// LS Electric XG5000 project: Villa 4 - ALS
// PLC NewPLC
// module base 0 slot 0: Input/Output Module:XBC-DR40S (DC 24V INPUT 24points/RELAY OUTPUT 16points)
// module base 0 slot 1: FEnet:XBL-EMTA

PROGRAM Main (task: Scan Program)

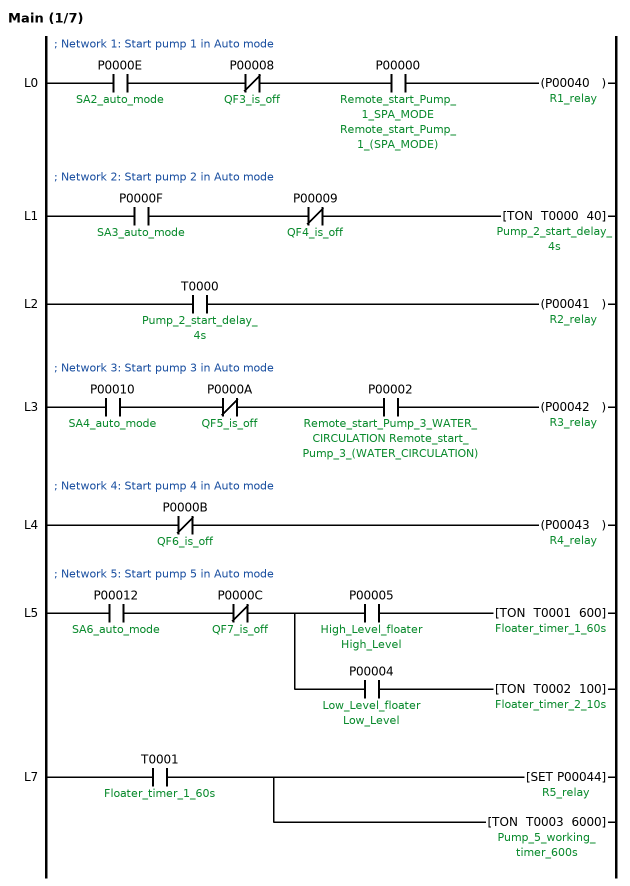
; L0
LOAD      P0000E	// SA2_auto_mode
AND NOT   P00008	// QF3_is_off
AND       P00000	// Remote_start_Pump_1_SPA_MODE Remote_start_Pump_1_(SPA_MODE)
OUT       P00040	// R1_relay
// output comment: Network 1: Start pump 1 in Auto mode
; L1
LOAD      P0000F	// SA3_auto_mode
AND NOT   P00009	// QF4_is_off
TON       T0000 40	// Pump_2_start_delay_4s
// output comment: Network 2: Start pump 2 in Auto mode
; L2
LOAD      T0000	// Pump_2_start_delay_4s
OUT       P00041	// R2_relay
; L3
LOAD      P00010	// SA4_auto_mode
AND NOT   P0000A	// QF5_is_off
AND       P00002	// Remote_start_Pump_3_WATER_CIRCULATION Remote_start_Pump_3_(WATER_CIRCULATION)
OUT       P00042	// R3_relay
// output comment: Network 3: Start pump 3 in Auto mode
; L4
LOAD NOT  P0000B	// QF6_is_off
OUT       P00043	// R4_relay
// output comment: Network 4: Start pump 4 in Auto mode
; L5
LOAD      P00012	// SA6_auto_mode
AND NOT   P0000C	// QF7_is_off
MPUSH
AND       P00005	// High_Level_floater High_Level
TON       T0001 600	// Floater_timer_1_60s
MPOP
AND       P00004	// Low_Level_floater Low_Level
TON       T0002 100	// Floater_timer_2_10s
// output comment: Network 5: Start pump 5 in Auto mode
; L7
LOAD      T0001	// Floater_timer_1_60s
SET       P00044	// R5_relay
TON       T0003 6000	// Pump_5_working_timer_600s

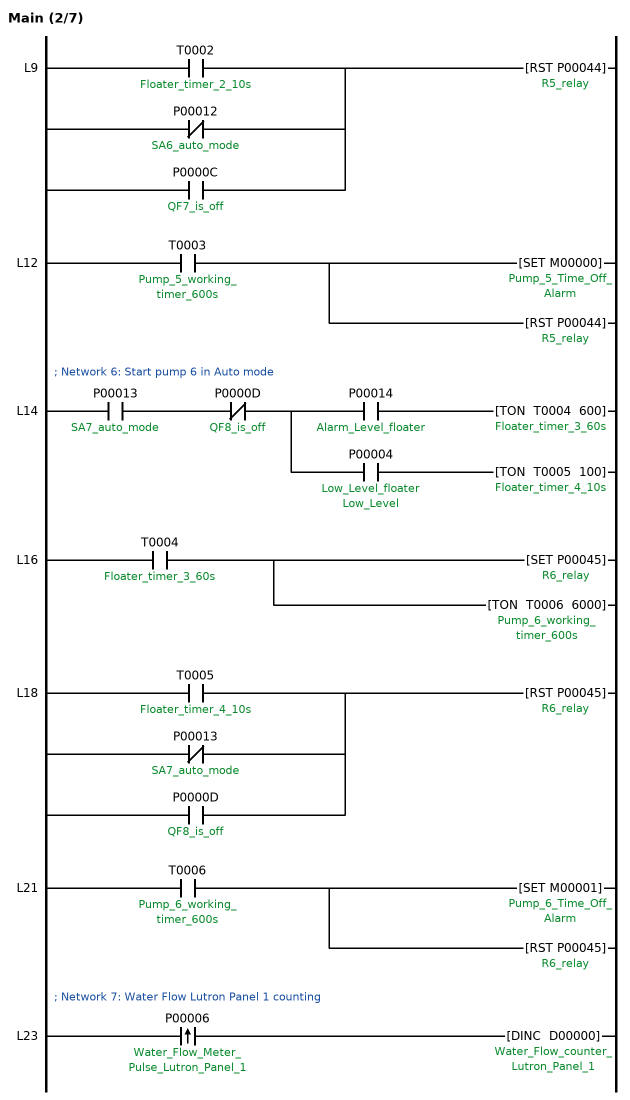
; L9
LOAD      T0002	// Floater_timer_2_10s
OR NOT    P00012	// SA6_auto_mode
OR        P0000C	// QF7_is_off
RST       P00044	// R5_relay
; L12
LOAD      T0003	// Pump_5_working_timer_600s
SET       M00000	// Pump_5_Time_Off_Alarm
RST       P00044	// R5_relay
; L14
LOAD      P00013	// SA7_auto_mode
AND NOT   P0000D	// QF8_is_off
MPUSH
AND       P00014	// Alarm_Level_floater
TON       T0004 600	// Floater_timer_3_60s
MPOP
AND       P00004	// Low_Level_floater Low_Level
TON       T0005 100	// Floater_timer_4_10s
// output comment: Network 6: Start pump 6 in Auto mode
; L16
LOAD      T0004	// Floater_timer_3_60s
SET       P00045	// R6_relay
TON       T0006 6000	// Pump_6_working_timer_600s
; L18
LOAD      T0005	// Floater_timer_4_10s
OR NOT    P00013	// SA7_auto_mode
OR        P0000D	// QF8_is_off
RST       P00045	// R6_relay
; L21
LOAD      T0006	// Pump_6_working_timer_600s
SET       M00001	// Pump_6_Time_Off_Alarm
RST       P00045	// R6_relay
; L23
LOADP     P00006	// Water_Flow_Meter_Pulse_Lutron_Panel_1
DINC      D00000	// Water_Flow_counter_Lutron_Panel_1
// output comment: Network 7: Water Flow Lutron Panel 1 counting

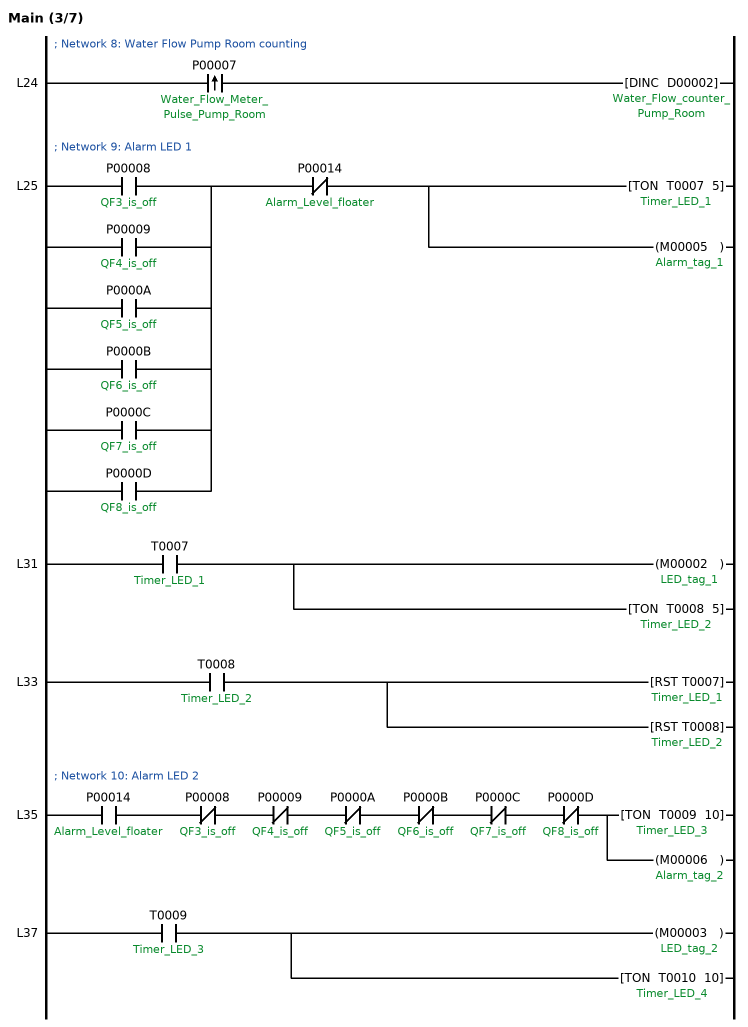
; L24
LOADP     P00007	// Water_Flow_Meter_Pulse_Pump_Room
DINC      D00002	// Water_Flow_counter_Pump_Room
// output comment: Network 8: Water Flow Pump Room counting
; L25
LOAD      P00008	// QF3_is_off
OR        P00009	// QF4_is_off
OR        P0000A	// QF5_is_off
OR        P0000B	// QF6_is_off
OR        P0000C	// QF7_is_off
OR        P0000D	// QF8_is_off
AND NOT   P00014	// Alarm_Level_floater
TON       T0007 5	// Timer_LED_1
OUT       M00005	// Alarm_tag_1
// output comment: Network 9: Alarm LED 1
; L31
LOAD      T0007	// Timer_LED_1
OUT       M00002	// LED_tag_1
TON       T0008 5	// Timer_LED_2
; L33
LOAD      T0008	// Timer_LED_2
RST       T0007	// Timer_LED_1
RST       T0008	// Timer_LED_2
; L35
LOAD      P00014	// Alarm_Level_floater
AND NOT   P00008	// QF3_is_off
AND NOT   P00009	// QF4_is_off
AND NOT   P0000A	// QF5_is_off
AND NOT   P0000B	// QF6_is_off
AND NOT   P0000C	// QF7_is_off
AND NOT   P0000D	// QF8_is_off
TON       T0009 10	// Timer_LED_3
OUT       M00006	// Alarm_tag_2
// output comment: Network 10: Alarm LED 2
; L37
LOAD      T0009	// Timer_LED_3
OUT       M00003	// LED_tag_2
TON       T0010 10	// Timer_LED_4

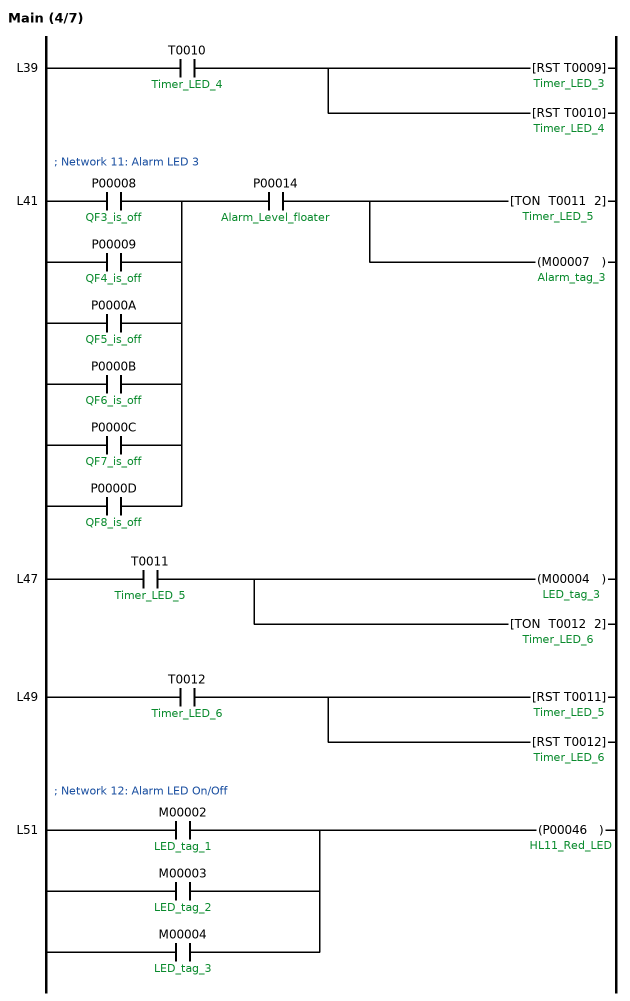
; L39
LOAD      T0010	// Timer_LED_4
RST       T0009	// Timer_LED_3
RST       T0010	// Timer_LED_4
; L41
LOAD      P00008	// QF3_is_off
OR        P00009	// QF4_is_off
OR        P0000A	// QF5_is_off
OR        P0000B	// QF6_is_off
OR        P0000C	// QF7_is_off
OR        P0000D	// QF8_is_off
AND       P00014	// Alarm_Level_floater
TON       T0011 2	// Timer_LED_5
OUT       M00007	// Alarm_tag_3
// output comment: Network 11: Alarm LED 3
; L47
LOAD      T0011	// Timer_LED_5
OUT       M00004	// LED_tag_3
TON       T0012 2	// Timer_LED_6
; L49
LOAD      T0012	// Timer_LED_6
RST       T0011	// Timer_LED_5
RST       T0012	// Timer_LED_6
; L51
LOAD      M00002	// LED_tag_1
OR        M00003	// LED_tag_2
OR        M00004	// LED_tag_3
OUT       P00046	// HL11_Red_LED
// output comment: Network 12: Alarm LED On/Off

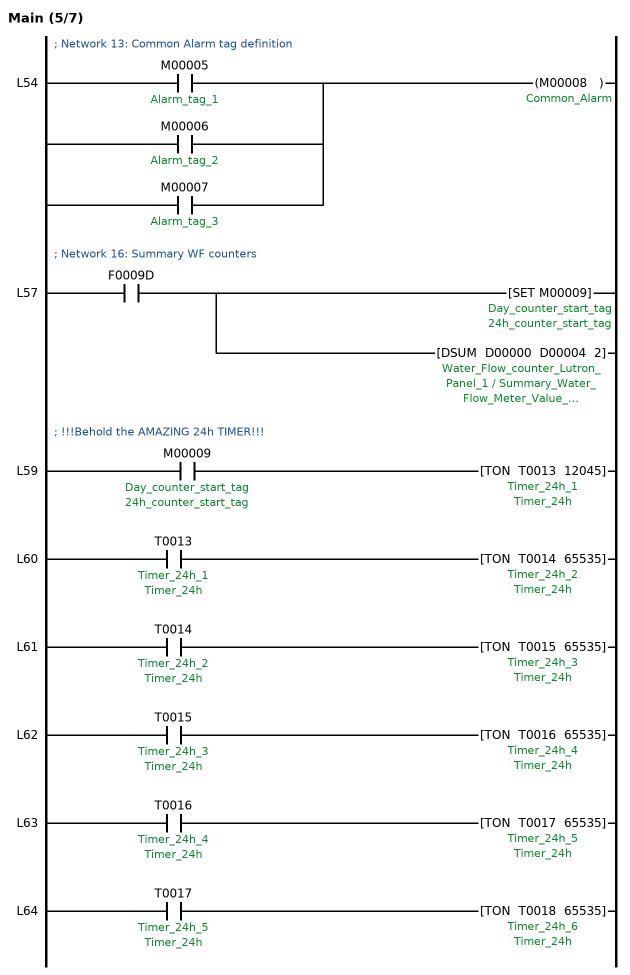
; L54
LOAD      M00005	// Alarm_tag_1
OR        M00006	// Alarm_tag_2
OR        M00007	// Alarm_tag_3
OUT       M00008	// Common_Alarm
// output comment: Network 13: Common Alarm tag definition
; L57
LOAD      F0009D
SET       M00009	// Day_counter_start_tag 24h_counter_start_tag
DSUM      D00000 D00004 2	// Water_Flow_counter_Lutron_Panel_1 / Summary_Water_Flow_Meter_Value_T Summary_Water_Flow_Meter_Value_(T)
// output comment: Network 16: Summary WF counters
; L59
LOAD      M00009	// Day_counter_start_tag 24h_counter_start_tag
TON       T0013 12045	// Timer_24h_1 Timer_24h
// output comment: !!!Behold the AMAZING 24h TIMER!!!
; L60
LOAD      T0013	// Timer_24h_1 Timer_24h
TON       T0014 65535	// Timer_24h_2 Timer_24h
; L61
LOAD      T0014	// Timer_24h_2 Timer_24h
TON       T0015 65535	// Timer_24h_3 Timer_24h
; L62
LOAD      T0015	// Timer_24h_3 Timer_24h
TON       T0016 65535	// Timer_24h_4 Timer_24h
; L63
LOAD      T0016	// Timer_24h_4 Timer_24h
TON       T0017 65535	// Timer_24h_5 Timer_24h
; L64
LOAD      T0017	// Timer_24h_5 Timer_24h
TON       T0018 65535	// Timer_24h_6 Timer_24h

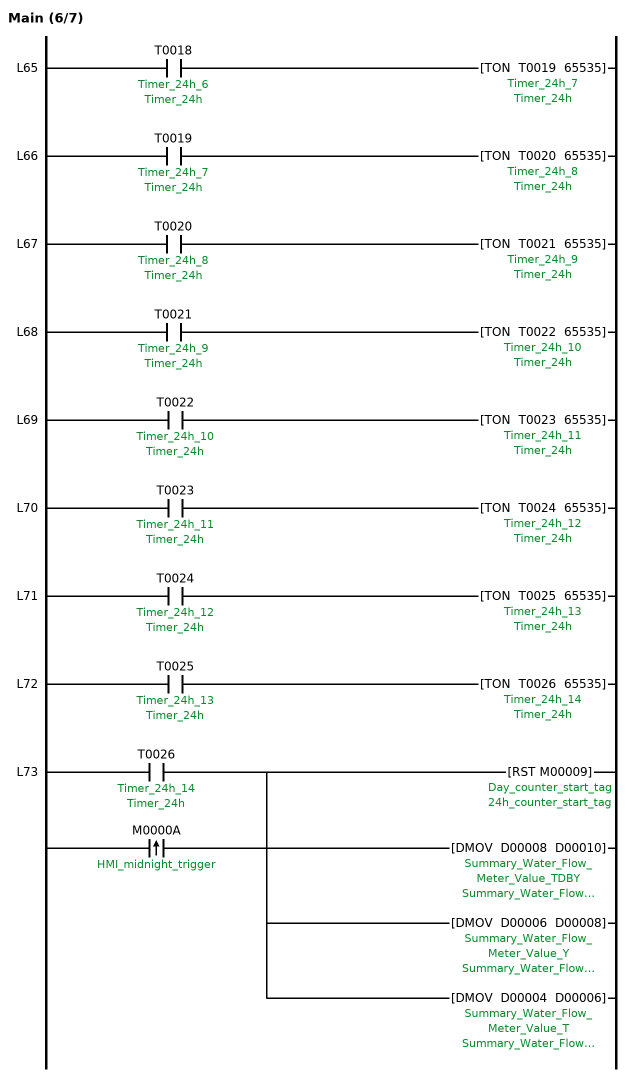
; L65
LOAD      T0018	// Timer_24h_6 Timer_24h
TON       T0019 65535	// Timer_24h_7 Timer_24h
; L66
LOAD      T0019	// Timer_24h_7 Timer_24h
TON       T0020 65535	// Timer_24h_8 Timer_24h
; L67
LOAD      T0020	// Timer_24h_8 Timer_24h
TON       T0021 65535	// Timer_24h_9 Timer_24h
; L68
LOAD      T0021	// Timer_24h_9 Timer_24h
TON       T0022 65535	// Timer_24h_10 Timer_24h
; L69
LOAD      T0022	// Timer_24h_10 Timer_24h
TON       T0023 65535	// Timer_24h_11 Timer_24h
; L70
LOAD      T0023	// Timer_24h_11 Timer_24h
TON       T0024 65535	// Timer_24h_12 Timer_24h
; L71
LOAD      T0024	// Timer_24h_12 Timer_24h
TON       T0025 65535	// Timer_24h_13 Timer_24h
; L72
LOAD      T0025	// Timer_24h_13 Timer_24h
TON       T0026 65535	// Timer_24h_14 Timer_24h
; L73
LOAD      T0026	// Timer_24h_14 Timer_24h
ORP       M0000A	// HMI_midnight_trigger
RST       M00009	// Day_counter_start_tag 24h_counter_start_tag
DMOV      D00008 D00010	// Summary_Water_Flow_Meter_Value_TDBY Summary_Water_Flow_Meter_Value_(TDBY) / Summary_Water_Flow_Meter_Value_TDBTDBY Summary_Water_Flow_Meter_Value_(TDBTDBY)
DMOV      D00006 D00008	// Summary_Water_Flow_Meter_Value_Y Summary_Water_Flow_Meter_Value_(Y) / Summary_Water_Flow_Meter_Value_TDBY Summary_Water_Flow_Meter_Value_(TDBY)
DMOV      D00004 D00006	// Summary_Water_Flow_Meter_Value_T Summary_Water_Flow_Meter_Value_(T) / Summary_Water_Flow_Meter_Value_Y Summary_Water_Flow_Meter_Value_(Y)

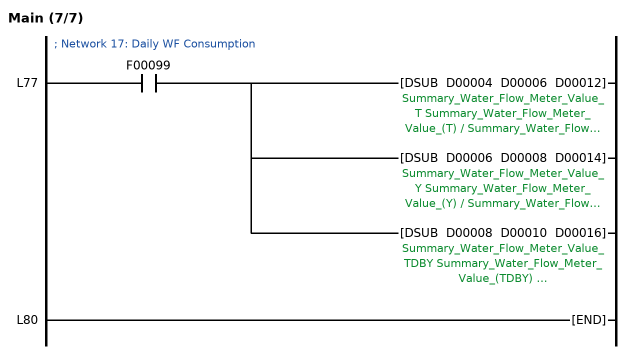
; L77
LOAD      F00099
DSUB      D00004 D00006 D00012	// Summary_Water_Flow_Meter_Value_T Summary_Water_Flow_Meter_Value_(T) / Summary_Water_Flow_Meter_Value_Y Summary_Water_Flow_Meter_Value_(Y) / Daily_WF_consumption_T Daily_WF_consumption_(T)
DSUB      D00006 D00008 D00014	// Summary_Water_Flow_Meter_Value_Y Summary_Water_Flow_Meter_Value_(Y) / Summary_Water_Flow_Meter_Value_TDBY Summary_Water_Flow_Meter_Value_(TDBY) / Daily_WF_consumption_Y Daily_WF_consumption_(Y)
DSUB      D00008 D00010 D00016	// Summary_Water_Flow_Meter_Value_TDBY Summary_Water_Flow_Meter_Value_(TDBY) / Summary_Water_Flow_Meter_Value_TDBTDBY Summary_Water_Flow_Meter_Value_(TDBTDBY) / Daily_WF_consumption_TDBY Daily_WF_consumption_(TDBY)
// output comment: Network 17: Daily WF Consumption
; L80
END

VARIABLES AND COMMENTS (devices not used above)
P00003	BIT	Remote_start_Air_Compressor
P00001	BIT	Remote_start_Pump_2
P00011	BIT	SA5_auto_mode